FUNCTION_BLOCK FB_ComplementaryFilter
VAR_INPUT
	// Accelerometer angle [unit]
	fAccAngle 		: LREAL;
	// Gyro roll angle rate [unit/s]
	fGyroRate		: LREAL;
	// Filter ratio [0..1]
	fFilterRatio 	: LREAL;
	// Step time [s]
	fStepTime 		: LREAL;
END_VAR
VAR_OUTPUT
	// Filtered angle [unit]
	fAngle 	: LREAL := 0.0;
END_VAR
VAR
END_VAR


// θ(t) = (1 − α) · θ(t)a + α · (θt−1 + ω(t)g · dt)

fAngle := (1.0 - fFilterRatio)*fAccAngle + fFilterRatio*(fAngle + fGyroRate*fStepTime);

END_FUNCTION_BLOCK

(* stored: Version 1.1.0.1, ProductVersion 3.1.4024.9
   POU FB_ComplementaryFilter: Id {4c62a9fc-15bd-490c-ab27-22af31fc4756}, SpecialFunc None *)
